FUNCTION_BLOCK FB_Market EXTENDS FB_Station
VAR
END_VAR

METHOD Marketing : INT
VAR
	stTempUnit				: ST_Unit;
	iTempIndex				: INT;
	iSold					: INT;
END_VAR
Marketing := 0;
IF iLastIndex > 0 THEN
	FOR iTempIndex := 1 TO iLastIndex BY 1 DO
		stTempUnit := stUnitArr[iTempIndex];
		IF stTempUnit.iProgress < 6 THEN
			stTempUnit.iProgress := stTempUnit.iProgress + 1;
			stUnitArr[iTempIndex] := stTempUnit;
		ELSE
			IF stTempUnit.eType = 0 THEN
				Marketing := Marketing + 8;
			ELSIF 
				stTempUnit.eType = 1 THEN
				Marketing := Marketing + 15;
			END_IF
			RemoveUnit(iTempIndex);
		END_IF
	END_FOR
END_IF
END_METHOD

END_FUNCTION_BLOCK

(* stored: Version 1.1.0.1, ProductVersion 3.1.4024.12
   POU FB_Market: Id {b4d1e01c-c244-4b7b-bec0-15476fe266bd}, SpecialFunc None
   Method Marketing: Id {69fe06ce-d9d3-4452-bfe5-9712f83a336b} *)
